FUNCTION_BLOCK FB_LightControl_KNX implements I_LightControl
VAR_INPUT
END_VAR
VAR_OUTPUT
END_VAR
VAR
END_VAR

{warning 'add method implementation'}
METHOD M_Reset : BOOL
END_METHOD

{warning 'add method implementation'}
METHOD M_Set : BOOL
END_METHOD

{warning 'add property implementation'}
PROPERTY nAddress : DINT
GET
END_GET
SET
END_SET
END_PROPERTY

{warning 'add property implementation'}
PROPERTY nIlluminance : REAL
GET
END_GET
SET
END_SET
END_PROPERTY

END_FUNCTION_BLOCK

(* stored: Version 1.1.0.1, ProductVersion 3.1.4022.18
   POU FB_LightControl_KNX: Id {4bfb8e24-26f0-46e7-ba09-dfaf10e3fea7}, SpecialFunc None
   Method M_Reset: Id {060e12cd-39cf-4221-89fd-edd7bb2e21d2}
   Method M_Set: Id {7d8ec49e-dc62-416f-9c79-9b6b11bcfe6f}
   Property nAddress: Id {f8bcdbf6-08f6-46c0-a28b-fcb41b814287}
   Get Get: Id {6c380f5e-0488-4ec5-b45d-b6f015a90661}
   Set Set: Id {f8d2898c-a8be-4b7e-823b-e60730ce811f}
   Property nIlluminance: Id {2e7a22a6-cb6d-43de-9202-f4effafa89f3}
   Get Get: Id {861defde-c3c9-443b-ab3f-417efb228dd0}
   Set Set: Id {d471587b-3b5a-4507-a541-c41bf27f3922} *)
